--- program Diecast14 (robot Fanuc M-20iA/35M) ---
  Smooth(1)
  Set speed (100.0 mm/s)
  Set Ref.: LASER_RTCP
  Set Tool: Diecast14
  Show Diecast14
  MoveJ 1 to (24.61, -120.07, 138.9) mm, rotated rx -157.35 ry 20.22 rz -39.64 deg; joints [168.243, -26.644, 169.501, 59.983, 90.075, -199.96]
  MoveL 2 to (24.61, -120.07, 138.9) mm, rotated rx -157.35 ry 20.22 rz -39.64 deg; joints [168.243, -26.644, 169.501, 59.983, 90.075, -199.96]
  MoveL 3 to (24.61, -70.07, 52.3) mm, rotated rx -157.35 ry 20.22 rz -39.64 deg; joints [163.685, -27.706, 172.293, 59.268, 84.781, -200.091]
  MoveL 4 to (24.61, -70.07, 52.3) mm, rotated rx -157.35 ry 20.22 rz -39.64 deg; joints [163.685, -27.706, 172.293, 59.268, 84.781, -200.091]
  Set speed (100.0 mm/s)
  MoveL 5 to (25.73, -70.23, 52.58) mm, rotated rx -157.35 ry 20.22 rz -39.64 deg; joints [163.716, -27.787, 172.261, 59.271, 84.824, -200.08]
  MoveL 6 to (26.86, -70.4, 52.87) mm, rotated rx -157.35 ry 20.22 rz -39.64 deg; joints [163.747, -27.868, 172.229, 59.274, 84.867, -200.068]
  MoveL 7 to (28.05, -70.52, 53.18) mm, rotated rx -157.32 ry 20.18 rz -39.53 deg; joints [163.78, -27.954, 172.199, 59.278, 84.911, -199.95]
  MoveL 8 to (29.25, -70.64, 53.4) mm, rotated rx -157.32 ry 20.18 rz -39.53 deg; joints [163.809, -28.042, 172.167, 59.28, 84.951, -199.937]
  MoveL 9 to (30.62, -70.63, 53.7) mm, rotated rx -157.22 ry 20.06 rz -39.24 deg; joints [163.844, -28.141, 172.141, 59.285, 84.994, -199.635]
  MoveL 10 to (31.68, -70.71, 53.84) mm, rotated rx -157.22 ry 20.06 rz -39.24 deg; joints [163.866, -28.219, 172.115, 59.287, 85.027, -199.624]
  MoveL 11 to (33.25, -69.4, 54.6) mm, rotated rx -156.34 ry 19 rz -36.62 deg; joints [163.924, -28.309, 172.18, 59.302, 85.042, -197.024]
  MoveL 12 to (34.48, -69.48, 54.74) mm, rotated rx -156.34 ry 19 rz -36.62 deg; joints [163.948, -28.401, 172.149, 59.304, 85.079, -197.01]
  MoveL 13 to (35.71, -69.55, 54.88) mm, rotated rx -156.34 ry 19 rz -36.62 deg; joints [163.973, -28.494, 172.118, 59.306, 85.115, -196.996]
  MoveL 14 to (39.02, -67.46, 56.27) mm, rotated rx -155.2 ry 17.45 rz -32.99 deg; joints [164.084, -28.696, 172.205, 59.333, 85.166, -193.349]
  MoveL 15 to (40.13, -67.52, 56.37) mm, rotated rx -155.2 ry 17.45 rz -32.99 deg; joints [164.104, -28.78, 172.177, 59.334, 85.198, -193.335]
  MoveL 16 to (41.24, -67.58, 56.47) mm, rotated rx -155.2 ry 17.45 rz -32.99 deg; joints [164.125, -28.864, 172.149, 59.336, 85.23, -193.322]
  MoveL 17 to (42.35, -67.64, 56.58) mm, rotated rx -155.2 ry 17.45 rz -32.99 deg; joints [164.146, -28.948, 172.121, 59.338, 85.261, -193.309]
  MoveL 18 to (44.51, -66.34, 57.46) mm, rotated rx -154.64 ry 16.58 rz -31.05 deg; joints [164.217, -29.082, 172.172, 59.354, 85.296, -191.342]
  MoveL 19 to (45.51, -66.38, 57.53) mm, rotated rx -154.64 ry 16.58 rz -31.05 deg; joints [164.235, -29.158, 172.147, 59.355, 85.324, -191.33]
  MoveL 20 to (46.51, -66.42, 57.6) mm, rotated rx -154.64 ry 16.58 rz -31.05 deg; joints [164.252, -29.235, 172.122, 59.357, 85.351, -191.317]
  MoveL 21 to (47.51, -66.46, 57.67) mm, rotated rx -154.64 ry 16.58 rz -31.05 deg; joints [164.269, -29.311, 172.098, 59.358, 85.379, -191.305]
  MoveL 22 to (49.02, -65.73, 58.19) mm, rotated rx -154.36 ry 16.13 rz -30.06 deg; joints [164.314, -29.41, 172.119, 59.367, 85.406, -190.293]
  MoveL 23 to (50.07, -65.75, 58.23) mm, rotated rx -154.36 ry 16.13 rz -30.06 deg; joints [164.331, -29.491, 172.094, 59.369, 85.433, -190.28]
  MoveL 24 to (51.11, -65.78, 58.28) mm, rotated rx -154.36 ry 16.13 rz -30.06 deg; joints [164.347, -29.571, 172.068, 59.37, 85.46, -190.266]
  MoveL 25 to (52.16, -65.8, 58.33) mm, rotated rx -154.36 ry 16.13 rz -30.06 deg; joints [164.364, -29.652, 172.042, 59.371, 85.487, -190.252]
  MoveL 26 to (53.2, -65.83, 58.37) mm, rotated rx -154.36 ry 16.13 rz -30.06 deg; joints [164.38, -29.733, 172.016, 59.372, 85.515, -190.239]
  MoveL 27 to (49.18, -71.56, 55.07) mm, rotated rx -156.5 ry 19.21 rz -37.11 deg; joints [164.176, -29.558, 171.678, 59.312, 85.513, -197.231]
  MoveL 28 to (50.38, -71.57, 55.09) mm, rotated rx -156.5 ry 19.21 rz -37.11 deg; joints [164.193, -29.652, 171.649, 59.314, 85.542, -197.215]
  MoveL 29 to (51.58, -71.58, 55.11) mm, rotated rx -156.5 ry 19.21 rz -37.11 deg; joints [164.211, -29.745, 171.621, 59.315, 85.572, -197.199]
  MoveL 30 to (52.78, -71.59, 55.13) mm, rotated rx -156.5 ry 19.21 rz -37.11 deg; joints [164.228, -29.839, 171.592, 59.316, 85.602, -197.183]
  MoveL 31 to (45.2, -79.81, 50.38) mm, rotated rx -160.52 ry 23.27 rz -48.16 deg; joints [163.909, -29.453, 171.146, 59.226, 85.558, -207.698]
  MoveL 32 to (46.6, -79.81, 50.38) mm, rotated rx -160.52 ry 23.27 rz -48.16 deg; joints [163.929, -29.563, 171.113, 59.228, 85.592, -207.68]
  MoveL 33 to (38.47, -86.11, 46.75) mm, rotated rx -164.82 ry 26.19 rz -58.43 deg; joints [163.649, -29.091, 170.82, 59.153, 85.504, -217.059]
  MoveL 34 to (39.84, -86.14, 46.81) mm, rotated rx -164.82 ry 26.19 rz -58.43 deg; joints [163.672, -29.197, 170.787, 59.156, 85.54, -217.042]
  MoveL 35 to (28.82, -92.99, 42.93) mm, rotated rx -171.39 ry 28.85 rz -72.58 deg; joints [163.337, -28.52, 170.513, 59.069, 85.398, -229.456]
  MoveL 36 to (30.3, -93.07, 43.07) mm, rotated rx -171.39 ry 28.85 rz -72.58 deg; joints [163.366, -28.633, 170.476, 59.073, 85.441, -229.439]
  MoveL 37 to (31.79, -93.15, 43.21) mm, rotated rx -171.39 ry 28.85 rz -72.58 deg; joints [163.395, -28.746, 170.439, 59.076, 85.485, -229.422]
  MoveL 38 to (12.32, -99.1, 39.78) mm, rotated rx 178.56 ry 29.97 rz -92.89 deg; joints [162.948, -27.403, 170.401, 58.98, 85.127, -246.863]
  MoveL 39 to (13.33, -99.1, 39.78) mm, rotated rx 178.56 ry 29.97 rz -92.89 deg; joints [162.964, -27.48, 170.38, 58.982, 85.151, -246.852]
  MoveL 40 to (14.33, -99.1, 39.78) mm, rotated rx 178.56 ry 29.97 rz -92.89 deg; joints [162.979, -27.557, 170.359, 58.984, 85.174, -246.842]
  MoveL 41 to (15.33, -99.1, 39.78) mm, rotated rx 178.56 ry 29.97 rz -92.89 deg; joints [162.994, -27.635, 170.339, 58.986, 85.198, -246.832]
  MoveL 42 to (16.34, -99.1, 39.78) mm, rotated rx 178.56 ry 29.97 rz -92.89 deg; joints [163.009, -27.712, 170.318, 58.987, 85.221, -246.822]
  MoveL 43 to (-9.54, -100.46, 38.99) mm, rotated rx 166.15 ry 26.88 rz -118.6 deg; joints [162.573, -25.777, 170.717, 58.926, 84.647, -269.718]
  MoveL 44 to (-8.53, -100.46, 38.99) mm, rotated rx 166.15 ry 26.88 rz -118.6 deg; joints [162.589, -25.853, 170.699, 58.928, 84.669, -269.71]
  MoveL 45 to (-7.53, -100.46, 38.99) mm, rotated rx 166.15 ry 26.88 rz -118.6 deg; joints [162.605, -25.929, 170.681, 58.93, 84.692, -269.703]
  MoveL 46 to (-6.53, -100.46, 38.99) mm, rotated rx 166.15 ry 26.88 rz -118.6 deg; joints [162.62, -26.005, 170.663, 58.932, 84.715, -269.695]
  MoveL 47 to (-5.52, -100.46, 38.99) mm, rotated rx 166.15 ry 26.88 rz -118.6 deg; joints [162.636, -26.08, 170.644, 58.933, 84.738, -269.687]
  MoveL 48 to (-22.4, -97.29, 40.83) mm, rotated rx 159.34 ry 22.25 rz -134.88 deg; joints [162.453, -24.731, 171.177, 58.939, 84.308, -285.551]
  MoveL 49 to (-20.57, -97.29, 40.83) mm, rotated rx 159.34 ry 22.25 rz -134.88 deg; joints [162.482, -24.866, 171.147, 58.943, 84.348, -285.54]
  MoveL 50 to (-31.87, -93.11, 43.24) mm, rotated rx 155.75 ry 18.23 rz -145.23 deg; joints [162.412, -23.922, 171.639, 58.972, 84.035, -296.432]
  MoveL 51 to (-30.87, -93.06, 43.14) mm, rotated rx 155.75 ry 18.23 rz -145.23 deg; joints [162.423, -23.997, 171.626, 58.973, 84.051, -296.427]
  MoveL 52 to (-29.87, -93, 43.04) mm, rotated rx 155.75 ry 18.23 rz -145.23 deg; joints [162.435, -24.073, 171.613, 58.974, 84.067, -296.422]
  MoveL 53 to (-41.24, -86.13, 46.88) mm, rotated rx 152.56 ry 12.62 rz -157.18 deg; joints [162.43, -23.072, 172.288, 59.035, 83.716, -309.813]
  MoveL 54 to (-39.89, -86.1, 46.83) mm, rotated rx 152.56 ry 12.62 rz -157.18 deg; joints [162.449, -23.172, 172.27, 59.037, 83.741, -309.808]
  MoveL 55 to (-38.53, -86.07, 46.77) mm, rotated rx 152.56 ry 12.62 rz -157.18 deg; joints [162.468, -23.272, 172.252, 59.039, 83.767, -309.802]
  MoveL 56 to (-46.6, -79.81, 50.38) mm, rotated rx 151 ry 8.02 rz -165.87 deg; joints [162.508, -22.536, 172.822, 59.101, 83.508, -320.017]
  MoveL 57 to (-45.2, -79.81, 50.38) mm, rotated rx 151 ry 8.02 rz -165.87 deg; joints [162.532, -22.639, 172.803, 59.103, 83.538, -320.012]
  MoveL 58 to (-52.78, -71.59, 55.13) mm, rotated rx 150.1 ry 2.57 rz -175.54 deg; joints [162.636, -21.904, 173.498, 59.191, 83.27, -331.728]
  MoveL 59 to (-51.58, -71.58, 55.11) mm, rotated rx 150.1 ry 2.57 rz -175.54 deg; joints [162.655, -21.992, 173.483, 59.192, 83.294, -331.725]
  MoveL 60 to (-50.38, -71.57, 55.09) mm, rotated rx 150.1 ry 2.57 rz -175.54 deg; joints [162.673, -22.079, 173.468, 59.194, 83.317, -331.721]
  MoveL 61 to (-49.18, -71.56, 55.07) mm, rotated rx 150.1 ry 2.57 rz -175.54 deg; joints [162.692, -22.167, 173.453, 59.196, 83.341, -331.718]
  MoveL 62 to (-53.13, -65.95, 58.3) mm, rotated rx 150.02 ry -1.05 rz 178.19 deg; joints [162.784, -21.762, 173.908, 59.258, 83.187, -339.398]
  MoveL 63 to (-52.02, -65.92, 58.25) mm, rotated rx 150.02 ry -1.05 rz 178.19 deg; joints [162.8, -21.842, 173.895, 59.259, 83.207, -339.395]
  MoveL 64 to (-50.92, -65.89, 58.2) mm, rotated rx 150.02 ry -1.05 rz 178.19 deg; joints [162.815, -21.923, 173.883, 59.26, 83.226, -339.392]
  MoveL 65 to (-49.82, -65.86, 58.14) mm, rotated rx 150.02 ry -1.05 rz 178.19 deg; joints [162.83, -22.004, 173.87, 59.261, 83.246, -339.389]
  MoveL 66 to (-48.71, -65.83, 58.09) mm, rotated rx 150.02 ry -1.05 rz 178.19 deg; joints [162.845, -22.085, 173.857, 59.263, 83.265, -339.386]
  MoveL 67 to (-46.68, -67.11, 57.28) mm, rotated rx 150 ry -0.12 rz 179.79 deg; joints [162.838, -22.262, 173.737, 59.249, 83.321, -337.43]
  MoveL 68 to (-45.54, -67.06, 57.18) mm, rotated rx 150 ry -0.12 rz 179.79 deg; joints [162.852, -22.346, 173.725, 59.25, 83.338, -337.426]
  MoveL 69 to (-44.41, -67.01, 57.09) mm, rotated rx 150 ry -0.12 rz 179.79 deg; joints [162.865, -22.43, 173.713, 59.251, 83.356, -337.423]
  MoveL 70 to (-43.27, -66.95, 57) mm, rotated rx 150 ry -0.12 rz 179.79 deg; joints [162.878, -22.515, 173.7, 59.252, 83.374, -337.419]
  MoveL 71 to (-42.13, -66.9, 56.9) mm, rotated rx 150 ry -0.12 rz 179.79 deg; joints [162.892, -22.599, 173.687, 59.253, 83.392, -337.414]
  MoveL 72 to (-38.77, -69.33, 55.38) mm, rotated rx 150.06 ry 1.94 rz -176.64 deg; joints [162.872, -22.9, 173.464, 59.228, 83.489, -333.085]
  MoveL 73 to (-37.75, -69.27, 55.27) mm, rotated rx 150.06 ry 1.94 rz -176.64 deg; joints [162.882, -22.976, 173.453, 59.229, 83.503, -333.081]
  MoveL 74 to (-36.73, -69.21, 55.15) mm, rotated rx 150.06 ry 1.94 rz -176.64 deg; joints [162.892, -23.052, 173.442, 59.229, 83.518, -333.076]
  MoveL 75 to (-35.71, -69.14, 55.04) mm, rotated rx 150.06 ry 1.94 rz -176.64 deg; joints [162.903, -23.129, 173.43, 59.23, 83.532, -333.072]
  MoveL 76 to (-34.7, -69.08, 54.93) mm, rotated rx 150.06 ry 1.94 rz -176.64 deg; joints [162.913, -23.205, 173.419, 59.231, 83.547, -333.067]
  MoveL 77 to (-33.68, -69.01, 54.82) mm, rotated rx 150.06 ry 1.94 rz -176.64 deg; joints [162.923, -23.282, 173.408, 59.231, 83.562, -333.063]
  MoveL 78 to (-31.55, -70.81, 53.79) mm, rotated rx 150.21 ry 3.75 rz -173.47 deg; joints [162.907, -23.477, 173.246, 59.213, 83.631, -329.269]
  MoveL 79 to (-30.4, -70.7, 53.59) mm, rotated rx 150.21 ry 3.75 rz -173.47 deg; joints [162.915, -23.565, 173.235, 59.213, 83.643, -329.264]
  MoveL 80 to (-29.25, -70.59, 53.4) mm, rotated rx 150.21 ry 3.75 rz -173.47 deg; joints [162.923, -23.653, 173.223, 59.213, 83.656, -329.258]
  MoveL 81 to (-27.98, -70.56, 53.15) mm, rotated rx 150.23 ry 3.85 rz -173.3 deg; joints [162.93, -23.751, 173.204, 59.213, 83.672, -329.044]
  MoveL 82 to (-26.86, -70.4, 52.87) mm, rotated rx 150.23 ry 3.85 rz -173.3 deg; joints [162.933, -23.839, 173.196, 59.213, 83.678, -329.039]
  MoveL 83 to (-25.73, -70.23, 52.58) mm, rotated rx 150.23 ry 3.85 rz -173.3 deg; joints [162.935, -23.927, 173.187, 59.212, 83.685, -329.032]
  MoveL 84 to (-24.61, -70.07, 52.3) mm, rotated rx 150.23 ry 3.85 rz -173.3 deg; joints [162.938, -24.015, 173.179, 59.212, 83.691, -329.026]
  Set speed (100.0 mm/s)
  MoveL 85 to (-24.61, -70.07, 52.3) mm, rotated rx 150.23 ry 3.85 rz -173.3 deg; joints [162.938, -24.015, 173.179, 59.212, 83.691, -329.026]
  MoveL 86 to (-5.32, -126.59, 135.13) mm, rotated rx 154.96 ry 17.09 rz -147.82 deg; joints [167.727, -24.481, 169.576, 59.889, 89.598, -300.047]
  Set speed (100.0 mm/s)
  MoveL 87 to (5.32, -126.59, 135.13) mm, rotated rx 154.96 ry 17.09 rz -147.82 deg; joints [167.847, -25.301, 169.387, 59.911, 89.795, -299.942]
  MoveL 88 to (5.32, -76.59, 48.53) mm, rotated rx 154.96 ry 17.09 rz -147.82 deg; joints [163.225, -26.396, 172.186, 59.175, 84.444, -300.04]
  MoveL 89 to (24.61, -70.07, 52.3) mm, rotated rx 165.93 ry 26.77 rz -119.09 deg; joints [163.685, -27.706, 172.293, 59.268, 84.781, -272.092]
  Set speed (100.0 mm/s)
  MoveL 90 to (25.73, -70.23, 52.58) mm, rotated rx 165.93 ry 26.77 rz -119.09 deg; joints [163.716, -27.787, 172.261, 59.271, 84.824, -272.08]
  MoveL 91 to (26.86, -70.4, 52.87) mm, rotated rx 165.93 ry 26.77 rz -119.09 deg; joints [163.747, -27.868, 172.229, 59.274, 84.867, -272.068]
  MoveL 92 to (28.05, -70.52, 53.18) mm, rotated rx 165.99 ry 26.8 rz -118.97 deg; joints [163.78, -27.954, 172.199, 59.278, 84.911, -271.95]
  MoveL 93 to (29.25, -70.64, 53.4) mm, rotated rx 165.99 ry 26.8 rz -118.97 deg; joints [163.809, -28.042, 172.167, 59.28, 84.951, -271.937]
  MoveL 94 to (30.62, -70.63, 53.7) mm, rotated rx 166.13 ry 26.87 rz -118.65 deg; joints [163.844, -28.141, 172.141, 59.285, 84.994, -271.635]
  MoveL 95 to (31.68, -70.71, 53.84) mm, rotated rx 166.13 ry 26.87 rz -118.65 deg; joints [163.866, -28.219, 172.115, 59.287, 85.027, -271.624]
  MoveL 96 to (33.25, -69.4, 54.6) mm, rotated rx 167.47 ry 27.48 rz -115.71 deg; joints [163.924, -28.309, 172.18, 59.302, 85.042, -269.024]
  MoveL 97 to (34.48, -69.48, 54.74) mm, rotated rx 167.47 ry 27.48 rz -115.71 deg; joints [163.948, -28.401, 172.149, 59.304, 85.079, -269.01]
  MoveL 98 to (35.71, -69.55, 54.88) mm, rotated rx 167.47 ry 27.48 rz -115.71 deg; joints [163.973, -28.494, 172.118, 59.306, 85.115, -268.996]
  MoveL 99 to (39.02, -67.46, 56.27) mm, rotated rx 169.43 ry 28.24 rz -111.52 deg; joints [164.084, -28.696, 172.205, 59.333, 85.166, -265.349]
  MoveL 100 to (40.13, -67.52, 56.37) mm, rotated rx 169.43 ry 28.24 rz -111.52 deg; joints [164.104, -28.78, 172.177, 59.334, 85.198, -265.335]
  MoveL 101 to (41.24, -67.58, 56.47) mm, rotated rx 169.43 ry 28.24 rz -111.52 deg; joints [164.125, -28.864, 172.149, 59.336, 85.23, -265.322]
  MoveL 102 to (42.35, -67.64, 56.58) mm, rotated rx 169.43 ry 28.24 rz -111.52 deg; joints [164.146, -28.948, 172.121, 59.338, 85.261, -265.309]
  MoveL 103 to (44.51, -66.34, 57.46) mm, rotated rx 170.52 ry 28.6 rz -109.23 deg; joints [164.217, -29.082, 172.172, 59.354, 85.296, -263.342]
  MoveL 104 to (45.51, -66.38, 57.53) mm, rotated rx 170.52 ry 28.6 rz -109.23 deg; joints [164.235, -29.158, 172.147, 59.355, 85.324, -263.33]
  MoveL 105 to (46.51, -66.42, 57.6) mm, rotated rx 170.52 ry 28.6 rz -109.23 deg; joints [164.252, -29.235, 172.122, 59.357, 85.351, -263.317]
  MoveL 106 to (47.51, -66.46, 57.67) mm, rotated rx 170.52 ry 28.6 rz -109.23 deg; joints [164.269, -29.311, 172.098, 59.358, 85.379, -263.305]
  MoveL 107 to (49.02, -65.73, 58.19) mm, rotated rx 171.09 ry 28.76 rz -108.05 deg; joints [164.314, -29.41, 172.119, 59.367, 85.406, -262.293]
  MoveL 108 to (50.07, -65.75, 58.23) mm, rotated rx 171.09 ry 28.76 rz -108.05 deg; joints [164.331, -29.491, 172.094, 59.369, 85.433, -262.28]
  MoveL 109 to (51.11, -65.78, 58.28) mm, rotated rx 171.09 ry 28.76 rz -108.05 deg; joints [164.347, -29.571, 172.068, 59.37, 85.46, -262.266]
  MoveL 110 to (52.16, -65.8, 58.33) mm, rotated rx 171.09 ry 28.76 rz -108.05 deg; joints [164.364, -29.652, 172.042, 59.371, 85.487, -262.252]
  MoveL 111 to (53.2, -65.83, 58.37) mm, rotated rx 171.09 ry 28.76 rz -108.05 deg; joints [164.38, -29.733, 172.016, 59.372, 85.515, -262.239]
  MoveL 112 to (49.18, -71.56, 55.07) mm, rotated rx 167.21 ry 27.37 rz -116.27 deg; joints [164.176, -29.558, 171.678, 59.312, 85.513, -269.231]
  MoveL 113 to (50.38, -71.57, 55.09) mm, rotated rx 167.21 ry 27.37 rz -116.27 deg; joints [164.193, -29.652, 171.649, 59.314, 85.542, -269.215]
  MoveL 114 to (51.58, -71.58, 55.11) mm, rotated rx 167.21 ry 27.37 rz -116.27 deg; joints [164.211, -29.745, 171.621, 59.315, 85.572, -269.199]
  MoveL 115 to (52.78, -71.59, 55.13) mm, rotated rx 167.21 ry 27.37 rz -116.27 deg; joints [164.228, -29.839, 171.592, 59.316, 85.602, -269.183]
  MoveL 116 to (45.2, -79.81, 50.38) mm, rotated rx 162.02 ry 24.43 rz -128.13 deg; joints [163.909, -29.453, 171.146, 59.226, 85.558, -279.698]
  MoveL 117 to (46.6, -79.81, 50.38) mm, rotated rx 162.02 ry 24.43 rz -128.13 deg; joints [163.929, -29.563, 171.113, 59.228, 85.592, -279.68]
  MoveL 118 to (38.47, -86.11, 46.75) mm, rotated rx 158.15 ry 21.09 rz -138.09 deg; joints [163.649, -29.091, 170.82, 59.153, 85.504, -289.059]
  MoveL 119 to (39.84, -86.14, 46.81) mm, rotated rx 158.15 ry 21.09 rz -138.09 deg; joints [163.672, -29.197, 170.787, 59.156, 85.54, -289.042]
  MoveL 120 to (28.82, -92.99, 42.93) mm, rotated rx 154.21 ry 15.89 rz -150.46 deg; joints [163.337, -28.52, 170.513, 59.069, 85.398, -301.456]
  MoveL 121 to (30.3, -93.07, 43.07) mm, rotated rx 154.21 ry 15.89 rz -150.46 deg; joints [163.366, -28.633, 170.476, 59.073, 85.441, -301.439]
  MoveL 122 to (31.79, -93.15, 43.21) mm, rotated rx 154.21 ry 15.89 rz -150.46 deg; joints [163.395, -28.746, 170.439, 59.076, 85.485, -301.422]
  MoveL 123 to (12.32, -99.1, 39.78) mm, rotated rx 150.91 ry 7.68 rz -166.5 deg; joints [162.948, -27.403, 170.401, 58.98, 85.127, -318.862]
  MoveL 124 to (13.33, -99.1, 39.78) mm, rotated rx 150.91 ry 7.68 rz -166.5 deg; joints [162.964, -27.48, 170.38, 58.982, 85.151, -318.853]
  MoveL 125 to (14.33, -99.1, 39.78) mm, rotated rx 150.91 ry 7.68 rz -166.5 deg; joints [162.979, -27.557, 170.359, 58.984, 85.174, -318.842]
  MoveL 126 to (15.33, -99.1, 39.78) mm, rotated rx 150.91 ry 7.68 rz -166.5 deg; joints [162.994, -27.635, 170.339, 58.986, 85.198, -318.832]
  MoveL 127 to (16.34, -99.1, 39.78) mm, rotated rx 150.91 ry 7.68 rz -166.5 deg; joints [163.009, -27.712, 170.318, 58.987, 85.221, -318.823]
  MoveL 128 to (-9.54, -100.46, 38.99) mm, rotated rx 150.2 ry -3.63 rz 173.69 deg; joints [162.573, -25.777, 170.717, 58.926, 84.647, -341.717]
  MoveL 129 to (-8.53, -100.46, 38.99) mm, rotated rx 150.2 ry -3.63 rz 173.69 deg; joints [162.589, -25.853, 170.699, 58.928, 84.669, -341.71]
  MoveL 130 to (-7.53, -100.46, 38.99) mm, rotated rx 150.2 ry -3.63 rz 173.69 deg; joints [162.605, -25.929, 170.681, 58.93, 84.692, -341.703]
  MoveL 131 to (-6.53, -100.46, 38.99) mm, rotated rx 150.2 ry -3.63 rz 173.69 deg; joints [162.62, -26.005, 170.663, 58.932, 84.715, -341.695]
  MoveL 132 to (-5.52, -100.46, 38.99) mm, rotated rx 150.2 ry -3.63 rz 173.69 deg; joints [162.636, -26.08, 170.644, 58.933, 84.738, -341.687]
  MoveL 133 to (-22.4, -97.29, 40.83) mm, rotated rx 151.97 ry -11.16 rz 160.02 deg; joints [162.453, -24.731, 171.177, 58.939, 84.308, -357.551]
  MoveL 134 to (-20.57, -97.29, 40.83) mm, rotated rx 151.97 ry -11.16 rz 160.02 deg; joints [162.482, -24.866, 171.147, 58.943, 84.348, -357.54]
  MoveL 135 to (-31.87, -93.11, 43.24) mm, rotated rx 154.23 ry -15.92 rz 150.38 deg; joints [162.412, -23.922, 171.639, 58.972, 84.035, -368.432]
  MoveL 136 to (-30.87, -93.06, 43.14) mm, rotated rx 154.23 ry -15.92 rz 150.39 deg; joints [162.423, -23.997, 171.626, 58.973, 84.051, -368.427]
  MoveL 137 to (-29.87, -93, 43.05) mm, rotated rx 154.23 ry -15.92 rz 150.38 deg; joints [162.435, -24.073, 171.613, 58.974, 84.067, -368.422]
  MoveL 138 to (-41.24, -86.13, 46.88) mm, rotated rx 158.18 ry -21.11 rz 138.02 deg; joints [162.43, -23.072, 172.288, 59.035, 83.716, -381.813]
  MoveL 139 to (-39.89, -86.1, 46.83) mm, rotated rx 158.18 ry -21.11 rz 138.02 deg; joints [162.449, -23.172, 172.27, 59.037, 83.741, -381.808]
  MoveL 140 to (-38.53, -86.07, 46.77) mm, rotated rx 158.18 ry -21.11 rz 138.02 deg; joints [162.468, -23.272, 172.252, 59.039, 83.767, -381.802]
  MoveL 141 to (-46.6, -79.81, 50.38) mm, rotated rx 162.02 ry -24.43 rz 128.13 deg; joints [162.508, -22.536, 172.822, 59.101, 83.508, -392.017]
  MoveL 142 to (-45.2, -79.81, 50.38) mm, rotated rx 162.02 ry -24.43 rz 128.13 deg; joints [162.532, -22.639, 172.803, 59.103, 83.538, -392.012]
  MoveL 143 to (-52.78, -71.59, 55.13) mm, rotated rx 167.21 ry -27.37 rz 116.27 deg; joints [162.636, -21.904, 173.498, 59.191, 83.27, -403.728]
  MoveL 144 to (-51.58, -71.58, 55.11) mm, rotated rx 167.21 ry -27.37 rz 116.27 deg; joints [162.655, -21.992, 173.483, 59.192, 83.294, -403.725]
  MoveL 145 to (-50.38, -71.57, 55.09) mm, rotated rx 167.21 ry -27.37 rz 116.27 deg; joints [162.673, -22.079, 173.468, 59.194, 83.317, -403.721]
  MoveL 146 to (-49.18, -71.56, 55.07) mm, rotated rx 167.21 ry -27.37 rz 116.27 deg; joints [162.692, -22.167, 173.453, 59.196, 83.341, -403.718]
  MoveL 147 to (-53.13, -65.95, 58.3) mm, rotated rx 171.01 ry -28.74 rz 108.21 deg; joints [162.784, -21.762, 173.908, 59.258, 83.187, -411.398]
  MoveL 148 to (-52.02, -65.92, 58.25) mm, rotated rx 171.01 ry -28.74 rz 108.21 deg; joints [162.8, -21.842, 173.895, 59.259, 83.207, -411.395]
  MoveL 149 to (-50.92, -65.89, 58.2) mm, rotated rx 171.01 ry -28.74 rz 108.21 deg; joints [162.815, -21.923, 173.883, 59.26, 83.226, -411.392]
  MoveL 150 to (-49.82, -65.86, 58.14) mm, rotated rx 171.01 ry -28.74 rz 108.21 deg; joints [162.83, -22.004, 173.87, 59.261, 83.246, -411.389]
  MoveL 151 to (-48.71, -65.83, 58.09) mm, rotated rx 171.01 ry -28.74 rz 108.21 deg; joints [162.845, -22.085, 173.857, 59.263, 83.265, -411.386]
  MoveL 152 to (-46.68, -67.11, 57.28) mm, rotated rx 170.02 ry -28.44 rz 110.29 deg; joints [162.838, -22.262, 173.737, 59.249, 83.321, -409.43]
  MoveL 153 to (-45.54, -67.06, 57.18) mm, rotated rx 170.02 ry -28.44 rz 110.29 deg; joints [162.852, -22.346, 173.725, 59.25, 83.338, -409.426]
  MoveL 154 to (-44.41, -67.01, 57.09) mm, rotated rx 170.02 ry -28.44 rz 110.29 deg; joints [162.865, -22.43, 173.713, 59.251, 83.356, -409.423]
  MoveL 155 to (-43.27, -66.95, 57) mm, rotated rx 170.02 ry -28.44 rz 110.29 deg; joints [162.878, -22.515, 173.7, 59.252, 83.374, -409.419]
  MoveL 156 to (-42.13, -66.9, 56.91) mm, rotated rx 170.02 ry -28.44 rz 110.29 deg; joints [162.892, -22.599, 173.687, 59.253, 83.392, -409.414]
  MoveL 157 to (-38.77, -69.33, 55.38) mm, rotated rx 167.86 ry -27.64 rz 114.88 deg; joints [162.872, -22.9, 173.464, 59.228, 83.489, -405.085]
  MoveL 158 to (-37.75, -69.27, 55.27) mm, rotated rx 167.86 ry -27.64 rz 114.88 deg; joints [162.882, -22.976, 173.453, 59.229, 83.503, -405.081]
  MoveL 159 to (-36.73, -69.21, 55.15) mm, rotated rx 167.86 ry -27.64 rz 114.88 deg; joints [162.892, -23.052, 173.442, 59.229, 83.518, -405.076]
  MoveL 160 to (-35.71, -69.14, 55.04) mm, rotated rx 167.86 ry -27.64 rz 114.88 deg; joints [162.903, -23.129, 173.43, 59.23, 83.532, -405.072]
  MoveL 161 to (-34.7, -69.08, 54.93) mm, rotated rx 167.86 ry -27.64 rz 114.88 deg; joints [162.913, -23.205, 173.419, 59.231, 83.547, -405.067]
  MoveL 162 to (-33.68, -69.01, 54.82) mm, rotated rx 167.86 ry -27.64 rz 114.88 deg; joints [162.923, -23.282, 173.408, 59.231, 83.562, -405.063]
  MoveL 163 to (-31.55, -70.81, 53.79) mm, rotated rx 166.03 ry -26.82 rz 118.87 deg; joints [162.907, -23.477, 173.246, 59.213, 83.631, -401.269]
  MoveL 164 to (-30.4, -70.7, 53.59) mm, rotated rx 166.03 ry -26.82 rz 118.87 deg; joints [162.915, -23.565, 173.235, 59.213, 83.643, -401.264]
  MoveL 165 to (-29.25, -70.59, 53.4) mm, rotated rx 166.03 ry -26.82 rz 118.87 deg; joints [162.923, -23.653, 173.223, 59.213, 83.656, -401.258]
  MoveL 166 to (-27.98, -70.56, 53.15) mm, rotated rx 165.93 ry -26.77 rz 119.09 deg; joints [162.93, -23.751, 173.204, 59.213, 83.672, -401.044]
  MoveL 167 to (-26.86, -70.4, 52.87) mm, rotated rx 165.93 ry -26.77 rz 119.09 deg; joints [162.933, -23.839, 173.196, 59.213, 83.678, -401.039]
  MoveL 168 to (-25.73, -70.23, 52.58) mm, rotated rx 165.93 ry -26.77 rz 119.09 deg; joints [162.935, -23.927, 173.187, 59.212, 83.685, -401.032]
  MoveL 169 to (-24.61, -70.07, 52.3) mm, rotated rx 165.93 ry -26.77 rz 119.09 deg; joints [162.938, -24.015, 173.179, 59.212, 83.691, -401.026]
  Set speed (100.0 mm/s)
  MoveL 170 to (-24.61, -70.07, 52.3) mm, rotated rx 165.93 ry -26.77 rz 119.09 deg; joints [162.938, -24.015, 173.179, 59.212, 83.691, -401.026]
  MoveL 171 to (-5.32, -126.59, 135.13) mm, rotated rx 154.96 ry -17.09 rz 147.82 deg; joints [167.727, -24.481, 169.576, 59.889, 89.598, -372.047]
  Set speed (100.0 mm/s)
  MoveL 172 to (5.32, -126.59, 135.13) mm, rotated rx 154.96 ry -17.09 rz 147.82 deg; joints [167.847, -25.301, 169.387, 59.911, 89.795, -371.942]
  MoveL 173 to (5.32, -76.59, 48.53) mm, rotated rx 154.96 ry -17.09 rz 147.82 deg; joints [163.225, -26.396, 172.186, 59.175, 84.444, -372.04]
  MoveL 174 to (24.61, -70.07, 52.3) mm, rotated rx 150.23 ry -3.85 rz 173.3 deg; joints [163.685, -27.706, 172.293, 59.268, 84.781, -344.092]
  Set speed (100.0 mm/s)
  MoveL 175 to (25.73, -70.23, 52.58) mm, rotated rx 150.23 ry -3.85 rz 173.3 deg; joints [163.716, -27.787, 172.261, 59.271, 84.824, -344.08]
  MoveL 176 to (26.86, -70.4, 52.87) mm, rotated rx 150.23 ry -3.85 rz 173.3 deg; joints [163.747, -27.868, 172.229, 59.274, 84.867, -344.068]
  MoveL 177 to (28.05, -70.52, 53.18) mm, rotated rx 150.22 ry -3.8 rz 173.4 deg; joints [163.78, -27.954, 172.199, 59.278, 84.911, -343.95]
  MoveL 178 to (29.25, -70.64, 53.4) mm, rotated rx 150.22 ry -3.8 rz 173.4 deg; joints [163.809, -28.042, 172.167, 59.28, 84.951, -343.937]
  MoveL 179 to (30.62, -70.63, 53.7) mm, rotated rx 150.2 ry -3.65 rz 173.65 deg; joints [163.844, -28.141, 172.141, 59.285, 84.994, -343.635]
  MoveL 180 to (31.68, -70.71, 53.84) mm, rotated rx 150.2 ry -3.65 rz 173.65 deg; joints [163.866, -28.219, 172.115, 59.287, 85.027, -343.624]
  MoveL 181 to (33.25, -69.4, 54.6) mm, rotated rx 150.08 ry -2.31 rz 175.98 deg; joints [163.924, -28.309, 172.18, 59.302, 85.042, -341.024]
  MoveL 182 to (34.48, -69.48, 54.74) mm, rotated rx 150.08 ry -2.31 rz 175.98 deg; joints [163.948, -28.401, 172.149, 59.304, 85.079, -341.01]
  MoveL 183 to (35.71, -69.56, 54.88) mm, rotated rx 150.08 ry -2.31 rz 175.98 deg; joints [163.973, -28.494, 172.118, 59.306, 85.115, -340.996]
  MoveL 184 to (39.02, -67.46, 56.27) mm, rotated rx 150 ry -0.43 rz 179.26 deg; joints [164.084, -28.696, 172.205, 59.333, 85.166, -337.349]
  MoveL 185 to (40.13, -67.52, 56.37) mm, rotated rx 150 ry -0.43 rz 179.26 deg; joints [164.104, -28.78, 172.177, 59.334, 85.198, -337.336]
  MoveL 186 to (41.24, -67.58, 56.47) mm, rotated rx 150 ry -0.43 rz 179.26 deg; joints [164.125, -28.864, 172.149, 59.336, 85.23, -337.322]
  MoveL 187 to (42.35, -67.64, 56.58) mm, rotated rx 150 ry -0.43 rz 179.26 deg; joints [164.146, -28.948, 172.121, 59.338, 85.261, -337.309]
  MoveL 188 to (44.51, -66.34, 57.46) mm, rotated rx 150.01 ry 0.6 rz -178.97 deg; joints [164.217, -29.082, 172.172, 59.354, 85.296, -335.342]
  MoveL 189 to (45.51, -66.38, 57.53) mm, rotated rx 150.01 ry 0.6 rz -178.97 deg; joints [164.235, -29.158, 172.147, 59.355, 85.324, -335.33]
  MoveL 190 to (46.51, -66.42, 57.6) mm, rotated rx 150.01 ry 0.6 rz -178.97 deg; joints [164.252, -29.235, 172.122, 59.357, 85.351, -335.317]
  MoveL 191 to (47.51, -66.46, 57.67) mm, rotated rx 150.01 ry 0.6 rz -178.97 deg; joints [164.269, -29.311, 172.098, 59.358, 85.379, -335.305]
  MoveL 192 to (49.02, -65.73, 58.19) mm, rotated rx 150.02 ry 1.12 rz -178.06 deg; joints [164.314, -29.41, 172.119, 59.367, 85.406, -334.293]
  MoveL 193 to (50.07, -65.75, 58.23) mm, rotated rx 150.02 ry 1.12 rz -178.06 deg; joints [164.331, -29.491, 172.094, 59.369, 85.433, -334.28]
  MoveL 194 to (51.11, -65.78, 58.28) mm, rotated rx 150.02 ry 1.12 rz -178.06 deg; joints [164.347, -29.571, 172.068, 59.37, 85.46, -334.266]
  MoveL 195 to (52.16, -65.8, 58.33) mm, rotated rx 150.02 ry 1.12 rz -178.06 deg; joints [164.364, -29.652, 172.042, 59.371, 85.487, -334.252]
  MoveL 196 to (53.2, -65.83, 58.37) mm, rotated rx 150.02 ry 1.12 rz -178.06 deg; joints [164.38, -29.733, 172.016, 59.372, 85.515, -334.238]
  MoveL 197 to (49.18, -71.56, 55.07) mm, rotated rx 150.1 ry -2.57 rz 175.54 deg; joints [164.176, -29.558, 171.678, 59.312, 85.513, -341.231]
  MoveL 198 to (50.38, -71.57, 55.09) mm, rotated rx 150.1 ry -2.57 rz 175.54 deg; joints [164.193, -29.652, 171.649, 59.314, 85.542, -341.215]
  MoveL 199 to (51.58, -71.58, 55.11) mm, rotated rx 150.1 ry -2.57 rz 175.54 deg; joints [164.211, -29.745, 171.621, 59.315, 85.572, -341.199]
  MoveL 200 to (52.78, -71.59, 55.13) mm, rotated rx 150.1 ry -2.57 rz 175.54 deg; joints [164.228, -29.839, 171.592, 59.316, 85.602, -341.183]
  MoveL 201 to (45.2, -79.81, 50.38) mm, rotated rx 151 ry -8.02 rz 165.87 deg; joints [163.909, -29.453, 171.146, 59.226, 85.558, -351.698]
  MoveL 202 to (46.6, -79.81, 50.38) mm, rotated rx 151 ry -8.02 rz 165.87 deg; joints [163.929, -29.563, 171.113, 59.228, 85.592, -351.68]
  MoveL 203 to (38.47, -86.11, 46.75) mm, rotated rx 152.57 ry -12.65 rz 157.12 deg; joints [163.649, -29.091, 170.82, 59.153, 85.504, -361.059]
  MoveL 204 to (39.84, -86.14, 46.81) mm, rotated rx 152.57 ry -12.65 rz 157.12 deg; joints [163.672, -29.197, 170.787, 59.156, 85.54, -361.042]
  MoveL 205 to (28.82, -92.99, 42.93) mm, rotated rx 155.77 ry -18.26 rz 145.15 deg; joints [163.337, -28.52, 170.513, 59.069, 85.398, -373.456]
  MoveL 206 to (30.3, -93.07, 43.07) mm, rotated rx 155.77 ry -18.26 rz 145.15 deg; joints [163.366, -28.633, 170.476, 59.073, 85.441, -373.439]
  MoveL 207 to (31.79, -93.15, 43.21) mm, rotated rx 155.77 ry -18.26 rz 145.15 deg; joints [163.395, -28.746, 170.439, 59.076, 85.485, -373.422]
  MoveL 208 to (12.32, -99.1, 39.78) mm, rotated rx 162.33 ry -24.64 rz 127.39 deg; joints [162.948, -27.403, 170.401, 58.98, 85.127, -390.862]
  MoveL 209 to (13.33, -99.1, 39.78) mm, rotated rx 162.33 ry -24.64 rz 127.39 deg; joints [162.964, -27.48, 170.38, 58.982, 85.151, -390.852]
  MoveL 210 to (14.33, -99.1, 39.78) mm, rotated rx 162.33 ry -24.64 rz 127.39 deg; joints [162.979, -27.557, 170.359, 58.984, 85.174, -390.843]
  MoveL 211 to (15.33, -99.1, 39.78) mm, rotated rx 162.33 ry -24.64 rz 127.39 deg; joints [162.994, -27.635, 170.339, 58.986, 85.198, -390.833]
  MoveL 212 to (16.34, -99.1, 39.78) mm, rotated rx 162.33 ry -24.64 rz 127.39 deg; joints [163.009, -27.712, 170.318, 58.987, 85.221, -390.822]
  MoveL 213 to (-9.54, -100.46, 38.99) mm, rotated rx 173.87 ry -29.42 rz 102.34 deg; joints [162.573, -25.777, 170.717, 58.926, 84.647, -413.717]
  MoveL 214 to (-8.53, -100.46, 38.99) mm, rotated rx 173.87 ry -29.42 rz 102.34 deg; joints [162.589, -25.853, 170.699, 58.928, 84.669, -413.71]
  MoveL 215 to (-7.53, -100.46, 38.99) mm, rotated rx 173.87 ry -29.42 rz 102.34 deg; joints [162.605, -25.929, 170.681, 58.93, 84.692, -413.703]
  MoveL 216 to (-6.53, -100.46, 38.99) mm, rotated rx 173.87 ry -29.42 rz 102.34 deg; joints [162.62, -26.005, 170.663, 58.932, 84.715, -413.695]
  MoveL 217 to (-5.52, -100.46, 38.99) mm, rotated rx 173.87 ry -29.42 rz 102.34 deg; joints [162.636, -26.08, 170.644, 58.933, 84.738, -413.687]
  MoveL 218 to (-22.4, -97.29, 40.83) mm, rotated rx -177.25 ry -29.89 rz 84.49 deg; joints [162.453, -24.731, 171.177, 58.939, 84.308, -429.551]
  MoveL 219 to (-20.57, -97.29, 40.83) mm, rotated rx -177.25 ry -29.89 rz 84.49 deg; joints [162.482, -24.866, 171.147, 58.943, 84.348, -429.54]
  MoveL 220 to (-31.87, -93.11, 43.24) mm, rotated rx -171.35 ry -28.84 rz 72.49 deg; joints [162.412, -23.922, 171.639, 58.972, 84.035, -440.432]
  MoveL 221 to (-30.87, -93.06, 43.14) mm, rotated rx -171.35 ry -28.84 rz 72.49 deg; joints [162.423, -23.997, 171.626, 58.973, 84.051, -440.427]
  MoveL 222 to (-29.87, -93, 43.04) mm, rotated rx -171.35 ry -28.84 rz 72.49 deg; joints [162.435, -24.073, 171.613, 58.974, 84.067, -440.422]
  MoveL 223 to (-9.29, -95.04, 46.88) mm, rotated rx -164.79 ry -26.17 rz 78.35 deg; joints [163.22, -26.8, 171.054, 64.59, 93.327, -435.869]
  MoveL 224 to (-8.03, -94.55, 46.83) mm, rotated rx -164.79 ry -26.17 rz 78.35 deg; joints [163.235, -26.891, 171.063, 64.592, 93.336, -435.884]
  MoveL 225 to (-6.77, -94.05, 46.77) mm, rotated rx -164.79 ry -26.17 rz 78.35 deg; joints [163.25, -26.982, 171.072, 64.593, 93.346, -435.898]
  MoveL 226 to (-16.5, -90.93, 50.38) mm, rotated rx -160.52 ry -23.27 rz 68.16 deg; joints [163.279, -26.123, 171.508, 64.574, 93.184, -446.007]
  MoveL 227 to (-15.17, -90.45, 50.38) mm, rotated rx -160.52 ry -23.27 rz 68.16 deg; joints [163.298, -26.218, 171.517, 64.576, 93.197, -446.023]
  MoveL 228 to (5.58, -88.77, 55.13) mm, rotated rx -156.5 ry -19.21 rz 77.11 deg; joints [164.033, -28.73, 171.554, 72.413, 100.174, -439.117]
  MoveL 229 to (6.5, -87.99, 55.11) mm, rotated rx -156.5 ry -19.21 rz 77.11 deg; joints [164.043, -28.792, 171.588, 72.408, 100.173, -439.153]
  MoveL 230 to (7.41, -87.21, 55.09) mm, rotated rx -156.5 ry -19.21 rz 77.11 deg; joints [164.052, -28.854, 171.622, 72.403, 100.172, -439.189]
  MoveL 231 to (8.32, -86.43, 55.07) mm, rotated rx -156.5 ry -19.21 rz 77.11 deg; joints [164.062, -28.916, 171.656, 72.398, 100.171, -439.225]
  MoveL 232 to (1.69, -84.67, 58.3) mm, rotated rx -154.4 ry -16.2 rz 70.2 deg; joints [164.127, -28.311, 171.954, 72.353, 100.141, -446.774]
  MoveL 233 to (2.52, -83.94, 58.25) mm, rotated rx -154.4 ry -16.2 rz 70.2 deg; joints [164.134, -28.368, 171.987, 72.348, 100.138, -446.808]
  MoveL 234 to (3.35, -83.2, 58.2) mm, rotated rx -154.4 ry -16.2 rz 70.2 deg; joints [164.141, -28.424, 172.02, 72.343, 100.135, -446.841]
  MoveL 235 to (4.17, -82.47, 58.14) mm, rotated rx -154.4 ry -16.2 rz 70.2 deg; joints [164.148, -28.481, 172.052, 72.338, 100.131, -446.875]
  MoveL 236 to (5, -81.74, 58.09) mm, rotated rx -154.4 ry -16.2 rz 70.2 deg; joints [164.155, -28.538, 172.084, 72.333, 100.128, -446.908]
  MoveL 237 to (7.38, -81.42, 57.28) mm, rotated rx -154.89 ry -16.99 rz 71.94 deg; joints [164.147, -28.737, 172.047, 72.339, 100.132, -445.021]
  MoveL 238 to (8.22, -80.65, 57.18) mm, rotated rx -154.89 ry -16.99 rz 71.94 deg; joints [164.152, -28.795, 172.081, 72.334, 100.126, -445.056]
  MoveL 239 to (9.05, -79.87, 57.09) mm, rotated rx -154.89 ry -16.99 rz 71.94 deg; joints [164.157, -28.853, 172.115, 72.328, 100.121, -445.091]
  MoveL 240 to (9.89, -79.1, 57) mm, rotated rx -154.89 ry -16.99 rz 71.94 deg; joints [164.162, -28.912, 172.149, 72.323, 100.115, -445.125]
  MoveL 241 to (10.73, -78.33, 56.91) mm, rotated rx -154.89 ry -16.99 rz 71.94 deg; joints [164.167, -28.97, 172.183, 72.317, 100.11, -445.16]
  MoveL 242 to (14.87, -78.03, 55.38) mm, rotated rx -156.1 ry -18.7 rz 75.89 deg; joints [164.148, -29.322, 172.095, 72.331, 100.118, -440.943]
  MoveL 243 to (15.61, -77.33, 55.27) mm, rotated rx -156.1 ry -18.7 rz 75.89 deg; joints [164.151, -29.374, 172.126, 72.326, 100.112, -440.974]
  MoveL 244 to (16.35, -76.63, 55.15) mm, rotated rx -156.1 ry -18.7 rz 75.89 deg; joints [164.154, -29.426, 172.157, 72.321, 100.105, -441.005]
  MoveL 245 to (17.08, -75.92, 55.04) mm, rotated rx -156.1 ry -18.7 rz 75.89 deg; joints [164.157, -29.479, 172.188, 72.316, 100.099, -441.035]
  MoveL 246 to (17.82, -75.22, 54.93) mm, rotated rx -156.1 ry -18.7 rz 75.89 deg; joints [164.16, -29.531, 172.218, 72.311, 100.092, -441.066]
  MoveL 247 to (18.56, -74.52, 54.82) mm, rotated rx -156.1 ry -18.7 rz 75.89 deg; joints [164.163, -29.583, 172.249, 72.306, 100.086, -441.097]
  MoveL 248 to (21.35, -74.53, 53.79) mm, rotated rx -157.28 ry -20.14 rz 79.44 deg; joints [164.15, -29.824, 172.173, 72.318, 100.097, -437.373]
  MoveL 249 to (22.15, -73.7, 53.59) mm, rotated rx -157.28 ry -20.14 rz 79.44 deg; joints [164.15, -29.882, 172.209, 72.312, 100.085, -437.408]
  MoveL 250 to (22.96, -72.88, 53.4) mm, rotated rx -157.28 ry -20.14 rz 79.44 deg; joints [164.149, -29.94, 172.246, 72.305, 100.074, -437.443]
  MoveL 251 to (23.92, -72.04, 53.15) mm, rotated rx -157.35 ry -20.22 rz 79.64 deg; joints [164.148, -30.011, 172.279, 72.3, 100.063, -437.275]
  MoveL 252 to (24.68, -71.19, 52.87) mm, rotated rx -157.35 ry -20.22 rz 79.64 deg; joints [164.142, -30.068, 172.317, 72.293, 100.046, -437.31]
  MoveL 253 to (25.43, -70.34, 52.58) mm, rotated rx -157.35 ry -20.22 rz 79.64 deg; joints [164.137, -30.124, 172.355, 72.286, 100.029, -437.345]
  MoveL 254 to (26.19, -69.49, 52.3) mm, rotated rx -157.35 ry -20.22 rz 79.64 deg; joints [164.131, -30.18, 172.393, 72.279, 100.012, -437.38]
  Set speed (100.0 mm/s)
  MoveL 255 to (26.19, -69.49, 52.3) mm, rotated rx -157.35 ry -20.22 rz 79.64 deg; joints [164.131, -30.18, 172.393, 72.279, 100.012, -437.38]
  MoveL 256 to (-5.32, -126.59, 135.13) mm, rotated rx -169.88 ry -28.39 rz 69.43 deg; joints [167.727, -24.481, 169.576, 59.889, 89.598, -444.047]
  Set speed (100.0 mm/s)
  MoveL 257 to (5.32, -126.59, 135.13) mm, rotated rx -169.88 ry -28.39 rz 69.43 deg; joints [167.847, -25.301, 169.387, 59.911, 89.795, -443.942]
  MoveL 258 to (5.32, -76.59, 48.53) mm, rotated rx -169.88 ry -28.39 rz 69.43 deg; joints [163.225, -26.396, 172.186, 59.175, 84.444, -444.04]
  MoveL 259 to (24.61, -70.07, 52.3) mm, rotated rx 174.12 ry -29.47 rz 101.82 deg; joints [163.685, -27.706, 172.293, 59.268, 84.781, -416.091]
  Set speed (100.0 mm/s)
  MoveL 260 to (25.73, -70.23, 52.58) mm, rotated rx 174.12 ry -29.47 rz 101.82 deg; joints [163.716, -27.787, 172.261, 59.271, 84.824, -416.08]
  MoveL 261 to (26.86, -70.4, 52.87) mm, rotated rx 174.12 ry -29.47 rz 101.82 deg; joints [163.747, -27.868, 172.229, 59.274, 84.867, -416.068]
  MoveL 262 to (28.05, -70.52, 53.18) mm, rotated rx 174.06 ry -29.46 rz 101.95 deg; joints [163.78, -27.954, 172.199, 59.278, 84.911, -415.95]
  MoveL 263 to (29.25, -70.64, 53.4) mm, rotated rx 174.06 ry -29.46 rz 101.95 deg; joints [163.809, -28.042, 172.167, 59.28, 84.951, -415.937]
  MoveL 264 to (30.62, -70.63, 53.7) mm, rotated rx 173.89 ry -29.43 rz 102.29 deg; joints [163.844, -28.141, 172.141, 59.285, 84.994, -415.635]
  MoveL 265 to (31.68, -70.71, 53.84) mm, rotated rx 173.89 ry -29.43 rz 102.29 deg; joints [163.866, -28.219, 172.115, 59.287, 85.027, -415.624]
  MoveL 266 to (33.25, -69.4, 54.6) mm, rotated rx 172.4 ry -29.11 rz 105.34 deg; joints [163.924, -28.309, 172.18, 59.302, 85.042, -413.024]
  MoveL 267 to (34.48, -69.48, 54.74) mm, rotated rx 172.4 ry -29.11 rz 105.34 deg; joints [163.948, -28.401, 172.149, 59.304, 85.079, -413.01]
  MoveL 268 to (35.71, -69.56, 54.88) mm, rotated rx 172.4 ry -29.11 rz 105.34 deg; joints [163.973, -28.494, 172.118, 59.306, 85.115, -412.996]
  MoveL 269 to (39.02, -67.46, 56.27) mm, rotated rx 170.34 ry -28.54 rz 109.61 deg; joints [164.084, -28.696, 172.205, 59.333, 85.166, -409.349]
  MoveL 270 to (40.13, -67.52, 56.37) mm, rotated rx 170.34 ry -28.54 rz 109.61 deg; joints [164.104, -28.78, 172.177, 59.334, 85.198, -409.335]
  MoveL 271 to (41.24, -67.58, 56.47) mm, rotated rx 170.34 ry -28.54 rz 109.61 deg; joints [164.125, -28.864, 172.149, 59.336, 85.23, -409.322]
  MoveL 272 to (42.35, -67.64, 56.58) mm, rotated rx 170.34 ry -28.54 rz 109.61 deg; joints [164.146, -28.948, 172.121, 59.338, 85.261, -409.309]
  MoveL 273 to (44.51, -66.34, 57.46) mm, rotated rx 169.25 ry -28.18 rz 111.89 deg; joints [164.217, -29.082, 172.172, 59.354, 85.296, -407.342]
  MoveL 274 to (45.51, -66.38, 57.53) mm, rotated rx 169.25 ry -28.18 rz 111.89 deg; joints [164.235, -29.158, 172.147, 59.355, 85.324, -407.33]
  MoveL 275 to (46.51, -66.42, 57.6) mm, rotated rx 169.25 ry -28.18 rz 111.89 deg; joints [164.252, -29.235, 172.122, 59.357, 85.351, -407.317]
  MoveL 276 to (47.51, -66.46, 57.67) mm, rotated rx 169.25 ry -28.18 rz 111.89 deg; joints [164.269, -29.311, 172.098, 59.358, 85.379, -407.305]
  MoveL 277 to (49.02, -65.73, 58.19) mm, rotated rx 168.7 ry -27.98 rz 113.07 deg; joints [164.314, -29.41, 172.119, 59.367, 85.406, -406.293]
  MoveL 278 to (50.07, -65.75, 58.23) mm, rotated rx 168.7 ry -27.98 rz 113.07 deg; joints [164.331, -29.491, 172.094, 59.369, 85.433, -406.28]
  MoveL 279 to (51.11, -65.78, 58.28) mm, rotated rx 168.7 ry -27.98 rz 113.07 deg; joints [164.347, -29.571, 172.068, 59.37, 85.46, -406.266]
  MoveL 280 to (52.16, -65.8, 58.33) mm, rotated rx 168.7 ry -27.98 rz 113.07 deg; joints [164.364, -29.652, 172.042, 59.371, 85.487, -406.252]
  MoveL 281 to (53.2, -65.83, 58.37) mm, rotated rx 168.7 ry -27.98 rz 113.07 deg; joints [164.38, -29.733, 172.016, 59.372, 85.515, -406.239]
  MoveL 282 to (49.18, -71.56, 55.07) mm, rotated rx 172.68 ry -29.17 rz 104.76 deg; joints [164.176, -29.558, 171.678, 59.312, 85.513, -413.231]
  MoveL 283 to (50.38, -71.57, 55.09) mm, rotated rx 172.68 ry -29.17 rz 104.76 deg; joints [164.193, -29.652, 171.649, 59.314, 85.542, -413.215]
  MoveL 284 to (51.58, -71.58, 55.11) mm, rotated rx 172.68 ry -29.17 rz 104.76 deg; joints [164.211, -29.745, 171.621, 59.315, 85.572, -413.199]
  MoveL 285 to (52.78, -71.59, 55.13) mm, rotated rx 172.68 ry -29.17 rz 104.76 deg; joints [164.228, -29.839, 171.592, 59.316, 85.602, -413.183]
  MoveL 286 to (45.2, -79.81, 50.38) mm, rotated rx 178.96 ry -29.98 rz 92.07 deg; joints [163.909, -29.453, 171.146, 59.226, 85.558, -423.698]
  MoveL 287 to (46.6, -79.81, 50.38) mm, rotated rx 178.96 ry -29.98 rz 92.07 deg; joints [163.929, -29.563, 171.113, 59.228, 85.592, -423.68]
  MoveL 288 to (38.47, -86.11, 46.75) mm, rotated rx -175.42 ry -29.68 rz 80.81 deg; joints [163.649, -29.091, 170.82, 59.153, 85.504, -433.059]
  MoveL 289 to (39.84, -86.14, 46.81) mm, rotated rx -175.42 ry -29.68 rz 80.81 deg; joints [163.672, -29.197, 170.787, 59.156, 85.54, -433.042]
  MoveL 290 to (28.82, -92.99, 42.93) mm, rotated rx -168.41 ry -27.87 rz 66.32 deg; joints [163.337, -28.52, 170.513, 59.069, 85.398, -445.456]
  MoveL 291 to (30.3, -93.07, 43.07) mm, rotated rx -168.41 ry -27.87 rz 66.32 deg; joints [163.366, -28.633, 170.476, 59.073, 85.441, -445.439]
  MoveL 292 to (31.79, -93.15, 43.21) mm, rotated rx -168.41 ry -27.87 rz 66.32 deg; joints [163.395, -28.746, 170.439, 59.076, 85.485, -445.422]
  MoveL 293 to (45.47, -88.91, 39.78) mm, rotated rx -160.23 ry -23.04 rz 67.43 deg; joints [163.648, -31.156, 170.177, 64.7, 94.084, -445.665]
  MoveL 294 to (46.42, -88.56, 39.78) mm, rotated rx -160.23 ry -23.04 rz 67.43 deg; joints [163.66, -31.227, 170.177, 64.701, 94.095, -445.67]
  MoveL 295 to (47.36, -88.22, 39.78) mm, rotated rx -160.23 ry -23.04 rz 67.43 deg; joints [163.673, -31.297, 170.177, 64.703, 94.106, -445.675]
  MoveL 296 to (48.3, -87.88, 39.78) mm, rotated rx -160.23 ry -23.04 rz 67.43 deg; joints [163.685, -31.368, 170.176, 64.705, 94.117, -445.68]
  MoveL 297 to (49.24, -87.54, 39.78) mm, rotated rx -160.23 ry -23.04 rz 67.43 deg; joints [163.697, -31.439, 170.176, 64.706, 94.128, -445.685]
  MoveL 298 to (82.23, -58.49, 38.99) mm, rotated rx -153.15 ry -13.9 rz 85.39 deg; joints [164.33, -35.62, 172.07, 81.85, 103.905, -432.768]
  MoveL 299 to (82.73, -57.62, 38.99) mm, rotated rx -153.15 ry -13.9 rz 85.39 deg; joints [164.335, -35.652, 172.116, 81.839, 103.902, -432.814]
  MoveL 300 to (83.24, -56.75, 38.99) mm, rotated rx -153.15 ry -13.9 rz 85.39 deg; joints [164.339, -35.683, 172.161, 81.828, 103.9, -432.861]
  MoveL 301 to (83.74, -55.88, 38.99) mm, rotated rx -153.15 ry -13.9 rz 85.39 deg; joints [164.344, -35.714, 172.207, 81.818, 103.898, -432.908]
  MoveL 302 to (84.24, -55.01, 38.99) mm, rotated rx -153.15 ry -13.9 rz 85.39 deg; joints [164.348, -35.746, 172.252, 81.807, 103.896, -432.955]
  MoveL 303 to (73.06, -68.04, 40.83) mm, rotated rx -150.66 ry -6.57 rz 71.5 deg; joints [164.32, -34.933, 171.706, 81.938, 103.945, -447.893]
  MoveL 304 to (73.97, -66.46, 40.83) mm, rotated rx -150.66 ry -6.57 rz 71.5 deg; joints [164.328, -34.989, 171.79, 81.918, 103.942, -447.98]
  MoveL 305 to (86.16, -47.55, 43.24) mm, rotated rx -150.03 ry -1.36 rz 82.36 deg; joints [164.591, -36.05, 173.72, 91.729, 104.491, -440.603]
  MoveL 306 to (86.28, -46.56, 43.14) mm, rotated rx -150.03 ry -1.36 rz 82.36 deg; joints [164.586, -36.053, 173.784, 91.711, 104.488, -440.669]
  MoveL 307 to (86.4, -45.56, 43.04) mm, rotated rx -150.03 ry -1.36 rz 82.36 deg; joints [164.581, -36.055, 173.849, 91.694, 104.485, -440.736]
  MoveL 308 to (91.98, -25.65, 46.88) mm, rotated rx -150.39 ry 5.03 rz 91.24 deg; joints [164.746, -36.156, 176.277, 101.023, 102.311, -436.359]
  MoveL 309 to (91.72, -24.33, 46.83) mm, rotated rx -150.39 ry 5.03 rz 91.24 deg; joints [164.737, -36.129, 176.374, 101.001, 102.321, -436.459]
  MoveL 310 to (91.45, -23, 46.77) mm, rotated rx -150.39 ry 5.03 rz 91.24 deg; joints [164.728, -36.102, 176.472, 100.979, 102.33, -436.558]
  MoveL 311 to (-86.69, 32.04, 50.38) mm, rotated rx -151.49 ry 9.75 rz -97.31 deg; joints [160.345, -15.976, 183.763, 79.318, 42.015, -266.682]
  MoveL 312 to (-45.2, -79.81, 50.38) mm, rotated rx -151.49 ry 9.75 rz -17.31 deg; joints [162.532, -22.639, 172.803, 59.103, 83.538, -176.012]
  MoveL 313 to (-52.78, -71.59, 55.13) mm, rotated rx -153.64 ry 14.86 rz -27.36 deg; joints [162.636, -21.904, 173.498, 59.191, 83.27, -187.728]
  MoveL 314 to (-51.58, -71.58, 55.11) mm, rotated rx -153.64 ry 14.86 rz -27.36 deg; joints [162.655, -21.992, 173.483, 59.192, 83.294, -187.725]
  MoveL 315 to (-50.38, -71.57, 55.09) mm, rotated rx -153.64 ry 14.86 rz -27.36 deg; joints [162.673, -22.079, 173.468, 59.194, 83.317, -187.721]
  MoveL 316 to (-49.18, -71.56, 55.07) mm, rotated rx -153.64 ry 14.86 rz -27.36 deg; joints [162.692, -22.167, 173.453, 59.196, 83.341, -187.718]
  MoveL 317 to (-53.13, -65.95, 58.3) mm, rotated rx -155.56 ry 17.97 rz -34.17 deg; joints [162.784, -21.762, 173.908, 59.258, 83.187, -195.398]
  MoveL 318 to (-52.02, -65.92, 58.25) mm, rotated rx -155.56 ry 17.97 rz -34.17 deg; joints [162.8, -21.842, 173.895, 59.259, 83.207, -195.395]
  MoveL 319 to (-50.92, -65.89, 58.2) mm, rotated rx -155.56 ry 17.97 rz -34.17 deg; joints [162.815, -21.923, 173.883, 59.26, 83.226, -195.392]
  MoveL 320 to (-49.82, -65.86, 58.14) mm, rotated rx -155.56 ry 17.97 rz -34.17 deg; joints [162.83, -22.004, 173.87, 59.261, 83.246, -195.389]
  MoveL 321 to (-48.71, -65.83, 58.09) mm, rotated rx -155.56 ry 17.97 rz -34.17 deg; joints [162.845, -22.085, 173.857, 59.263, 83.265, -195.386]
  MoveL 322 to (-46.68, -67.11, 57.28) mm, rotated rx -155.03 ry 17.2 rz -32.41 deg; joints [162.838, -22.262, 173.737, 59.249, 83.321, -193.43]
  MoveL 323 to (-45.54, -67.06, 57.18) mm, rotated rx -155.03 ry 17.2 rz -32.41 deg; joints [162.852, -22.346, 173.725, 59.25, 83.338, -193.426]
  MoveL 324 to (-44.41, -67.01, 57.09) mm, rotated rx -155.03 ry 17.2 rz -32.41 deg; joints [162.865, -22.43, 173.713, 59.251, 83.356, -193.422]
  MoveL 325 to (-43.27, -66.95, 57) mm, rotated rx -155.03 ry 17.2 rz -32.41 deg; joints [162.878, -22.515, 173.7, 59.252, 83.374, -193.419]
  MoveL 326 to (-42.13, -66.9, 56.9) mm, rotated rx -155.03 ry 17.2 rz -32.41 deg; joints [162.892, -22.599, 173.687, 59.253, 83.392, -193.414]
  MoveL 327 to (-38.77, -69.33, 55.38) mm, rotated rx -153.94 ry 15.42 rz -28.53 deg; joints [162.872, -22.9, 173.464, 59.228, 83.489, -189.085]
  MoveL 328 to (-37.75, -69.27, 55.27) mm, rotated rx -153.94 ry 15.42 rz -28.53 deg; joints [162.882, -22.976, 173.453, 59.229, 83.503, -189.081]
  MoveL 329 to (-36.73, -69.21, 55.15) mm, rotated rx -153.94 ry 15.42 rz -28.53 deg; joints [162.892, -23.052, 173.442, 59.229, 83.518, -189.077]
  MoveL 330 to (-35.71, -69.14, 55.04) mm, rotated rx -153.94 ry 15.42 rz -28.53 deg; joints [162.903, -23.129, 173.43, 59.23, 83.532, -189.072]
  MoveL 331 to (-34.7, -69.08, 54.93) mm, rotated rx -153.94 ry 15.42 rz -28.53 deg; joints [162.913, -23.205, 173.419, 59.231, 83.547, -189.067]
  MoveL 332 to (-33.68, -69.01, 54.82) mm, rotated rx -153.94 ry 15.42 rz -28.53 deg; joints [162.923, -23.282, 173.408, 59.231, 83.562, -189.063]
  MoveL 333 to (-31.55, -70.81, 53.79) mm, rotated rx -153.09 ry 13.79 rz -25.16 deg; joints [162.907, -23.477, 173.246, 59.213, 83.631, -185.269]
  MoveL 334 to (-30.4, -70.7, 53.59) mm, rotated rx -153.09 ry 13.79 rz -25.16 deg; joints [162.915, -23.565, 173.235, 59.213, 83.643, -185.264]
  MoveL 335 to (-29.25, -70.59, 53.4) mm, rotated rx -153.09 ry 13.79 rz -25.16 deg; joints [162.923, -23.653, 173.223, 59.213, 83.656, -185.258]
  MoveL 336 to (-27.98, -70.56, 53.15) mm, rotated rx -153.05 ry 13.7 rz -24.98 deg; joints [162.93, -23.751, 173.204, 59.213, 83.672, -185.044]
  MoveL 337 to (-26.86, -70.4, 52.87) mm, rotated rx -153.05 ry 13.7 rz -24.98 deg; joints [162.933, -23.839, 173.196, 59.213, 83.678, -185.039]
  MoveL 338 to (-25.73, -70.23, 52.58) mm, rotated rx -153.05 ry 13.7 rz -24.98 deg; joints [162.935, -23.927, 173.187, 59.212, 83.685, -185.032]
  MoveL 339 to (-24.61, -70.07, 52.3) mm, rotated rx -153.05 ry 13.7 rz -24.98 deg; joints [162.938, -24.015, 173.179, 59.212, 83.691, -185.026]
  Set speed (100.0 mm/s)
  MoveL 340 to (-24.61, -70.07, 52.3) mm, rotated rx -153.05 ry 13.7 rz -24.98 deg; joints [162.938, -24.015, 173.179, 59.212, 83.691, -185.026]
  MoveL 341 to (-5.32, -126.59, 135.13) mm, rotated rx -150 ry 0 rz 0 deg; joints [167.727, -24.481, 169.576, 59.889, 89.598, -156.047]
  Set speed (100.0 mm/s)
  MoveL 342 to (5.32, -126.59, 135.13) mm, rotated rx -150 ry 0 rz 0 deg; joints [167.847, -25.301, 169.387, 59.911, 89.795, -155.942]
  MoveL 343 to (5.32, -76.59, 48.53) mm, rotated rx -150 ry 0 rz 0 deg; joints [163.225, -26.396, 172.186, 59.175, 84.444, -156.04]
  MoveL 344 to (24.61, -70.07, 52.3) mm, rotated rx -153.05 ry -13.7 rz 24.98 deg; joints [163.685, -27.706, 172.293, 59.268, 84.781, -128.092]
  Set speed (100.0 mm/s)
  MoveL 345 to (25.73, -70.23, 52.58) mm, rotated rx -153.05 ry -13.7 rz 24.98 deg; joints [163.716, -27.787, 172.261, 59.271, 84.824, -128.08]
  MoveL 346 to (26.86, -70.4, 52.87) mm, rotated rx -153.05 ry -13.7 rz 24.98 deg; joints [163.747, -27.868, 172.229, 59.274, 84.867, -128.068]
  MoveL 347 to (28.05, -70.52, 53.18) mm, rotated rx -153.07 ry -13.75 rz 25.08 deg; joints [163.78, -27.954, 172.199, 59.278, 84.911, -127.95]
  MoveL 348 to (29.25, -70.64, 53.4) mm, rotated rx -153.07 ry -13.75 rz 25.08 deg; joints [163.809, -28.042, 172.167, 59.28, 84.951, -127.937]
  MoveL 349 to (30.62, -70.63, 53.7) mm, rotated rx -153.14 ry -13.88 rz 25.35 deg; joints [163.844, -28.141, 172.141, 59.285, 84.994, -127.635]
  MoveL 350 to (31.68, -70.71, 53.84) mm, rotated rx -153.14 ry -13.88 rz 25.35 deg; joints [163.866, -28.219, 172.115, 59.287, 85.027, -127.624]
  MoveL 351 to (33.25, -69.4, 54.6) mm, rotated rx -153.76 ry -15.09 rz 27.83 deg; joints [163.924, -28.309, 172.18, 59.302, 85.042, -125.024]
  MoveL 352 to (34.48, -69.48, 54.74) mm, rotated rx -153.76 ry -15.09 rz 27.83 deg; joints [163.948, -28.401, 172.149, 59.304, 85.079, -125.01]
  MoveL 353 to (35.71, -69.56, 54.88) mm, rotated rx -153.76 ry -15.09 rz 27.83 deg; joints [163.973, -28.494, 172.118, 59.306, 85.115, -124.996]
  MoveL 354 to (39.02, -67.46, 56.27) mm, rotated rx -154.73 ry -16.73 rz 31.37 deg; joints [164.084, -28.696, 172.205, 59.333, 85.166, -121.349]
  MoveL 355 to (40.13, -67.52, 56.37) mm, rotated rx -154.73 ry -16.73 rz 31.37 deg; joints [164.104, -28.78, 172.177, 59.334, 85.198, -121.335]
  MoveL 356 to (41.24, -67.58, 56.47) mm, rotated rx -154.73 ry -16.73 rz 31.37 deg; joints [164.125, -28.864, 172.149, 59.336, 85.23, -121.322]
  MoveL 357 to (42.35, -67.64, 56.58) mm, rotated rx -154.73 ry -16.73 rz 31.37 deg; joints [164.146, -28.948, 172.121, 59.338, 85.261, -121.309]
  MoveL 358 to (44.51, -66.34, 57.46) mm, rotated rx -155.3 ry -17.59 rz 33.31 deg; joints [164.217, -29.082, 172.172, 59.354, 85.296, -119.343]
  MoveL 359 to (45.51, -66.38, 57.53) mm, rotated rx -155.3 ry -17.59 rz 33.31 deg; joints [164.235, -29.158, 172.147, 59.355, 85.324, -119.33]
  MoveL 360 to (46.51, -66.42, 57.6) mm, rotated rx -155.3 ry -17.59 rz 33.31 deg; joints [164.252, -29.235, 172.122, 59.357, 85.351, -119.317]
  MoveL 361 to (47.51, -66.46, 57.67) mm, rotated rx -155.3 ry -17.59 rz 33.31 deg; joints [164.269, -29.311, 172.098, 59.358, 85.379, -119.305]
  MoveL 362 to (49.02, -65.73, 58.19) mm, rotated rx -155.61 ry -18.03 rz 34.32 deg; joints [164.314, -29.41, 172.119, 59.367, 85.406, -118.293]
  MoveL 363 to (50.07, -65.75, 58.23) mm, rotated rx -155.61 ry -18.03 rz 34.32 deg; joints [164.331, -29.491, 172.094, 59.369, 85.433, -118.28]
  MoveL 364 to (51.11, -65.78, 58.28) mm, rotated rx -155.61 ry -18.03 rz 34.32 deg; joints [164.347, -29.571, 172.068, 59.37, 85.46, -118.266]
  MoveL 365 to (52.16, -65.8, 58.33) mm, rotated rx -155.61 ry -18.03 rz 34.32 deg; joints [164.364, -29.652, 172.042, 59.371, 85.487, -118.252]
  MoveL 366 to (53.2, -65.83, 58.37) mm, rotated rx -155.61 ry -18.03 rz 34.32 deg; joints [164.38, -29.733, 172.016, 59.372, 85.515, -118.239]
  MoveL 367 to (49.18, -71.56, 55.07) mm, rotated rx -153.64 ry -14.86 rz 27.36 deg; joints [164.176, -29.558, 171.678, 59.312, 85.513, -125.231]
  MoveL 368 to (50.38, -71.57, 55.09) mm, rotated rx -153.64 ry -14.86 rz 27.36 deg; joints [164.193, -29.652, 171.649, 59.314, 85.542, -125.215]
  MoveL 369 to (51.58, -71.58, 55.11) mm, rotated rx -153.64 ry -14.86 rz 27.36 deg; joints [164.211, -29.745, 171.621, 59.315, 85.572, -125.199]
  MoveL 370 to (52.78, -71.59, 55.13) mm, rotated rx -153.64 ry -14.86 rz 27.36 deg; joints [164.228, -29.839, 171.592, 59.316, 85.602, -125.183]
  MoveL 371 to (45.2, -79.81, 50.38) mm, rotated rx -151.49 ry -9.75 rz 17.31 deg; joints [163.909, -29.453, 171.146, 59.226, 85.558, -135.698]
  MoveL 372 to (46.6, -79.81, 50.38) mm, rotated rx -151.49 ry -9.75 rz 17.31 deg; joints [163.929, -29.563, 171.113, 59.228, 85.592, -135.68]
  MoveL 373 to (38.47, -86.11, 46.75) mm, rotated rx -150.38 ry -4.99 rz 8.7 deg; joints [163.649, -29.091, 170.82, 59.153, 85.504, -145.059]
  MoveL 374 to (39.84, -86.14, 46.81) mm, rotated rx -150.38 ry -4.99 rz 8.7 deg; joints [163.672, -29.197, 170.787, 59.156, 85.54, -145.042]
  MoveL 375 to (28.82, -92.99, 42.93) mm, rotated rx -150.03 ry 1.4 rz -2.43 deg; joints [163.337, -28.52, 170.513, 59.069, 85.398, -157.456]
  MoveL 376 to (30.3, -93.07, 43.07) mm, rotated rx -150.03 ry 1.4 rz -2.43 deg; joints [163.366, -28.633, 170.476, 59.073, 85.441, -157.439]
  MoveL 377 to (31.79, -93.15, 43.21) mm, rotated rx -150.03 ry 1.4 rz -2.43 deg; joints [163.395, -28.746, 170.439, 59.076, 85.485, -157.422]
  MoveL 378 to (12.32, -99.1, 39.78) mm, rotated rx -151.6 ry 10.09 rz -17.94 deg; joints [162.948, -27.403, 170.401, 58.98, 85.127, -174.862]
  MoveL 379 to (13.33, -99.1, 39.78) mm, rotated rx -151.6 ry 10.09 rz -17.94 deg; joints [162.964, -27.48, 170.38, 58.982, 85.151, -174.852]
  MoveL 380 to (14.33, -99.1, 39.78) mm, rotated rx -151.6 ry 10.09 rz -17.94 deg; joints [162.979, -27.557, 170.359, 58.984, 85.174, -174.842]
  MoveL 381 to (15.33, -99.1, 39.78) mm, rotated rx -151.6 ry 10.09 rz -17.94 deg; joints [162.994, -27.635, 170.339, 58.986, 85.198, -174.832]
  MoveL 382 to (16.34, -99.1, 39.78) mm, rotated rx -151.6 ry 10.09 rz -17.94 deg; joints [163.009, -27.712, 170.318, 58.987, 85.221, -174.822]
  MoveL 383 to (-9.54, -100.46, 38.99) mm, rotated rx -157.2 ry 20.04 rz -39.19 deg; joints [162.573, -25.777, 170.717, 58.926, 84.647, -197.718]
  MoveL 384 to (-8.53, -100.46, 38.99) mm, rotated rx -157.2 ry 20.04 rz -39.19 deg; joints [162.589, -25.853, 170.699, 58.928, 84.669, -197.71]
  MoveL 385 to (-7.53, -100.46, 38.99) mm, rotated rx -157.2 ry 20.04 rz -39.19 deg; joints [162.605, -25.929, 170.681, 58.93, 84.692, -197.702]
  MoveL 386 to (-6.53, -100.46, 38.99) mm, rotated rx -157.2 ry 20.04 rz -39.19 deg; joints [162.62, -26.005, 170.663, 58.932, 84.715, -197.695]
  MoveL 387 to (-5.52, -100.46, 38.99) mm, rotated rx -157.2 ry 20.04 rz -39.19 deg; joints [162.636, -26.08, 170.644, 58.933, 84.738, -197.687]
  MoveL 388 to (-22.4, -97.29, 40.83) mm, rotated rx -163.34 ry 25.31 rz -55.01 deg; joints [162.453, -24.731, 171.177, 58.939, 84.308, -213.551]
  MoveL 389 to (-20.57, -97.29, 40.83) mm, rotated rx -163.34 ry 25.31 rz -55.01 deg; joints [162.482, -24.866, 171.147, 58.943, 84.348, -213.54]
  MoveL 390 to (-31.87, -93.11, 43.24) mm, rotated rx -168.45 ry 27.88 rz -66.4 deg; joints [162.412, -23.922, 171.639, 58.972, 84.035, -224.432]
  MoveL 391 to (-30.87, -93.06, 43.14) mm, rotated rx -168.45 ry 27.88 rz -66.4 deg; joints [162.423, -23.997, 171.626, 58.973, 84.051, -224.427]
  MoveL 392 to (-29.87, -93, 43.05) mm, rotated rx -168.45 ry 27.88 rz -66.4 deg; joints [162.435, -24.073, 171.613, 58.974, 84.067, -224.422]
  MoveL 393 to (-41.24, -86.13, 46.88) mm, rotated rx -175.46 ry 29.69 rz -80.89 deg; joints [162.43, -23.072, 172.288, 59.035, 83.716, -237.813]
  MoveL 394 to (-39.89, -86.1, 46.83) mm, rotated rx -175.46 ry 29.69 rz -80.89 deg; joints [162.449, -23.172, 172.27, 59.037, 83.741, -237.808]
  MoveL 395 to (-38.53, -86.07, 46.77) mm, rotated rx -175.46 ry 29.69 rz -80.89 deg; joints [162.468, -23.272, 172.252, 59.039, 83.767, -237.802]
  MoveL 396 to (-46.6, -79.81, 50.38) mm, rotated rx 178.96 ry 29.98 rz -92.07 deg; joints [162.508, -22.536, 172.822, 59.101, 83.508, -248.017]
  MoveL 397 to (-45.2, -79.81, 50.38) mm, rotated rx 178.96 ry 29.98 rz -92.07 deg; joints [162.532, -22.639, 172.803, 59.103, 83.538, -248.012]
  MoveL 398 to (-52.78, -71.59, 55.13) mm, rotated rx 172.68 ry 29.17 rz -104.76 deg; joints [162.636, -21.904, 173.498, 59.191, 83.27, -259.728]
  MoveL 399 to (-51.58, -71.58, 55.11) mm, rotated rx 172.68 ry 29.17 rz -104.76 deg; joints [162.655, -21.992, 173.483, 59.192, 83.294, -259.725]
  MoveL 400 to (-50.38, -71.57, 55.09) mm, rotated rx 172.68 ry 29.17 rz -104.76 deg; joints [162.673, -22.079, 173.468, 59.194, 83.317, -259.721]
  MoveL 401 to (-49.18, -71.56, 55.07) mm, rotated rx 172.68 ry 29.17 rz -104.76 deg; joints [162.692, -22.167, 173.453, 59.196, 83.341, -259.718]
  MoveL 402 to (-53.13, -65.95, 58.3) mm, rotated rx 168.78 ry 28.01 rz -112.9 deg; joints [162.785, -21.762, 173.908, 59.258, 83.187, -267.398]
  MoveL 403 to (-52.02, -65.92, 58.25) mm, rotated rx 168.78 ry 28.01 rz -112.9 deg; joints [162.8, -21.842, 173.895, 59.259, 83.207, -267.395]
  MoveL 404 to (-50.92, -65.89, 58.2) mm, rotated rx 168.78 ry 28.01 rz -112.9 deg; joints [162.815, -21.923, 173.883, 59.26, 83.226, -267.392]
  MoveL 405 to (-49.82, -65.86, 58.14) mm, rotated rx 168.78 ry 28.01 rz -112.9 deg; joints [162.83, -22.004, 173.87, 59.261, 83.246, -267.389]
  MoveL 406 to (-48.71, -65.83, 58.09) mm, rotated rx 168.78 ry 28.01 rz -112.9 deg; joints [162.845, -22.085, 173.857, 59.263, 83.265, -267.386]
  MoveL 407 to (-46.68, -67.11, 57.28) mm, rotated rx 169.75 ry 28.35 rz -110.84 deg; joints [162.838, -22.262, 173.737, 59.249, 83.321, -265.43]
  MoveL 408 to (-45.54, -67.06, 57.18) mm, rotated rx 169.75 ry 28.35 rz -110.84 deg; joints [162.852, -22.346, 173.725, 59.25, 83.338, -265.426]
  MoveL 409 to (-44.41, -67.01, 57.09) mm, rotated rx 169.75 ry 28.35 rz -110.84 deg; joints [162.865, -22.43, 173.713, 59.251, 83.356, -265.423]
  MoveL 410 to (-43.27, -66.95, 57) mm, rotated rx 169.75 ry 28.35 rz -110.84 deg; joints [162.878, -22.515, 173.7, 59.252, 83.374, -265.418]
  MoveL 411 to (-42.13, -66.9, 56.91) mm, rotated rx 169.75 ry 28.35 rz -110.84 deg; joints [162.892, -22.599, 173.687, 59.253, 83.392, -265.414]
  MoveL 412 to (-38.77, -69.33, 55.38) mm, rotated rx 171.98 ry 29.01 rz -106.2 deg; joints [162.872, -22.9, 173.464, 59.228, 83.489, -261.085]
  MoveL 413 to (-37.75, -69.27, 55.27) mm, rotated rx 171.98 ry 29.01 rz -106.2 deg; joints [162.882, -22.976, 173.453, 59.229, 83.503, -261.081]
  MoveL 414 to (-36.73, -69.21, 55.15) mm, rotated rx 171.98 ry 29.01 rz -106.2 deg; joints [162.892, -23.052, 173.442, 59.229, 83.518, -261.076]
  MoveL 415 to (-35.71, -69.14, 55.04) mm, rotated rx 171.98 ry 29.01 rz -106.2 deg; joints [162.903, -23.129, 173.43, 59.23, 83.532, -261.072]
  MoveL 416 to (-34.7, -69.08, 54.93) mm, rotated rx 171.98 ry 29.01 rz -106.2 deg; joints [162.913, -23.205, 173.419, 59.231, 83.547, -261.068]
  MoveL 417 to (-33.68, -69.01, 54.82) mm, rotated rx 171.98 ry 29.01 rz -106.2 deg; joints [162.923, -23.282, 173.408, 59.231, 83.562, -261.063]
  MoveL 418 to (-31.55, -70.81, 53.79) mm, rotated rx 174.01 ry 29.45 rz -102.05 deg; joints [162.907, -23.477, 173.246, 59.213, 83.631, -257.269]
  MoveL 419 to (-30.4, -70.7, 53.59) mm, rotated rx 174.01 ry 29.45 rz -102.05 deg; joints [162.915, -23.565, 173.235, 59.213, 83.643, -257.264]
  MoveL 420 to (-29.25, -70.59, 53.4) mm, rotated rx 174.01 ry 29.45 rz -102.05 deg; joints [162.923, -23.653, 173.223, 59.213, 83.656, -257.258]
  MoveL 421 to (-27.98, -70.56, 53.15) mm, rotated rx 174.12 ry 29.47 rz -101.82 deg; joints [162.93, -23.751, 173.204, 59.213, 83.672, -257.044]
  MoveL 422 to (-26.86, -70.4, 52.87) mm, rotated rx 174.12 ry 29.47 rz -101.82 deg; joints [162.933, -23.839, 173.196, 59.213, 83.678, -257.038]
  MoveL 423 to (-25.73, -70.23, 52.58) mm, rotated rx 174.12 ry 29.47 rz -101.82 deg; joints [162.935, -23.927, 173.187, 59.212, 83.685, -257.032]
  MoveL 424 to (-24.61, -70.07, 52.3) mm, rotated rx 174.12 ry 29.47 rz -101.82 deg; joints [162.938, -24.015, 173.179, 59.212, 83.691, -257.026]
  Set speed (100.0 mm/s)
  MoveL 425 to (-24.61, -70.07, 52.3) mm, rotated rx 174.12 ry 29.47 rz -101.82 deg; joints [162.938, -24.015, 173.179, 59.212, 83.691, -257.026]
  MoveL 426 to (-24.61, -120.07, 138.9) mm, rotated rx 174.12 ry 29.47 rz -101.82 deg; joints [167.694, -22.856, 170.364, 59.891, 89.175, -256.987]
